FUNCTION_BLOCK GOODFEATURESTOTRACK (* openCV goodFeaturesToTrack *)
  (* Version 1.0, AN, SWDC RTSoft *)
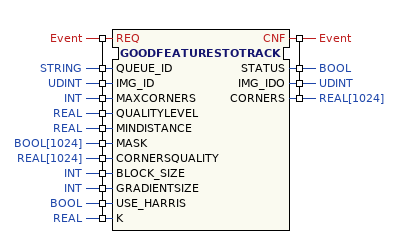
  EVENT_INPUT
    REQ WITH QUEUE_ID, IMG_ID, MAXCORNERS, QUALITYLEVEL, MINDISTANCE, MASK, CORNERSQUALITY, BLOCK_SIZE, GRADIENTSIZE, USE_HARRIS, K;
  END_EVENT
  EVENT_OUTPUT
    CNF WITH STATUS, IMG_IDO, CORNERS;
  END_EVENT
  VAR_INPUT
    QUEUE_ID : STRING;
    IMG_ID : UDINT;
    MAXCORNERS : INT; (* Maximum number of corners to return *)
    QUALITYLEVEL : REAL;
    MINDISTANCE : REAL; (* Minimum distance between returned corners *)
    MASK : ARRAY [0..1023] OF BOOL;
    CORNERSQUALITY : ARRAY [0..1023] OF REAL; (* Output vector for corner qualities *)
    BLOCK_SIZE : INT; (* Size of an average block for computing a derivative covariation matrix *)
    GRADIENTSIZE : INT;
    USE_HARRIS : BOOL;
    K : REAL; (* Harris detector free parameter *)
  END_VAR
  VAR_OUTPUT
    STATUS : BOOL;
    IMG_IDO : UDINT;
    CORNERS : ARRAY [0..1023] OF REAL;
  END_VAR
  ALGORITHM REQ IN ST:

  END_ALGORITHM
END_FUNCTION_BLOCK
